(* CoDeSys 2.3 export: J1939.EXP *)

(* POU J1939, ST *)
PROGRAM J1939
VAR CONSTANT
	Cycle_Time1 : REAL := 0.005; (*5ms*)
END_VAR
VAR
END_VAR
PARAMS; (*To Load Faster*)

(**********)
(* ENGINE *)
(**********)
RECV_J1939;
SEND_J1939;
END_PROGRAM
